FUNCTION_BLOCK INI_ALR2 (* Load and Store LREAL Data from settings.ini by Section and Key (ALR2 Adapter Interface) *)
  (* Standard: 61499-2; Description: Copyright (c) 2026 Meisterschulen am Ostbahnhof This program and the accompanying materials are made available under the terms of the Eclipse Public License 2.0 which is available at https://www.eclipse.org/legal/epl-2.0/ SPDX-License-Identifier: EPL-2.0 *)
  (* Version 1.0, 2026-09-12, Franz Höpfinger, Meisterschulen am Ostbahnhof, initial implementation - INI-Adapterfamilie vervollstaendigt (analog zu bestehenden INI_AX2/INI_AR2/INI_AB2). *)
  PACKAGE eclipse4diac::storage;
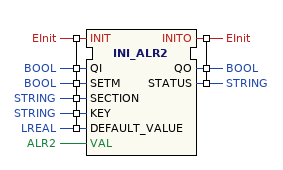
  EVENT_INPUT
    INIT : EInit WITH QI, SETM, SECTION, KEY, DEFAULT_VALUE; (* Service Initialization *)
  END_EVENT
  EVENT_OUTPUT
    INITO : EInit WITH QO, STATUS; (* Initialization Confirm *)
  END_EVENT
  VAR_INPUT
    QI : BOOL; (* Event Input Qualifier *)
    SETM : BOOL; (* Enable Mirroring on SET *)
    SECTION : STRING; (* Section name. *)
    KEY : STRING; (* Key name. *)
    DEFAULT_VALUE : LREAL; (* The value to read if there is nothing in the settings.ini *)
  END_VAR
  VAR_OUTPUT
    QO : BOOL; (* Event Output Qualifier *)
    STATUS : STRING; (* Service Status *)
  END_VAR
  SOCKETS
    VAL : adapter::types::bidirectional::ALR2; (* Value *)
  END_SOCKETS
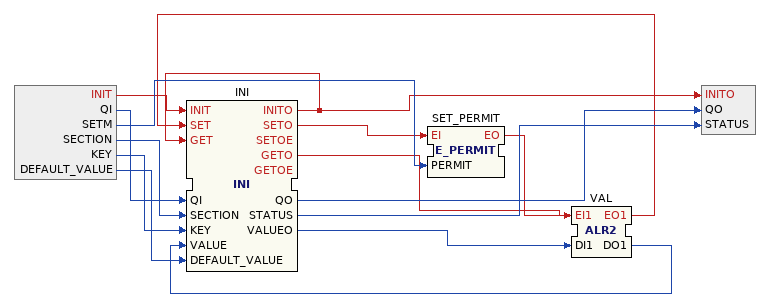
  FBS
    INI : eclipse4diac::storage::INI;
    SET_PERMIT : iec61499::events::E_PERMIT;
  END_FBS
  EVENT_CONNECTIONS
    INI.INITO TO INITO;
    INI.INITO TO INI.GET;
    VAL.EO1 TO INI.SET;
    SET_PERMIT.EO TO VAL.EI1;
    INI.GETO TO VAL.EI1;
    INIT TO INI.INIT;
    INI.SETO TO SET_PERMIT.EI;
  END_CONNECTIONS
  DATA_CONNECTIONS
    QI TO INI.QI;
    SETM TO SET_PERMIT.PERMIT;
    KEY TO INI.KEY;
    DEFAULT_VALUE TO INI.DEFAULT_VALUE;
    VAL.DO1 TO INI.VALUE;
    INI.VALUEO TO VAL.DI1;
    SECTION TO INI.SECTION;
    INI.STATUS TO STATUS;
    INI.QO TO QO;
  END_CONNECTIONS
END_FUNCTION_BLOCK
